        global vpPlaceStack2= pose_trans (pStackOutBase2_p, p[0,0,-1*iStackOut2*fSampleDoneZ,0,0,0])
        $ 1379 "PlaceStackOut"
        $ 1380 "If iStackOut1≤iStackOut2"
        if (iStackOut1 <= iStackOut2):
          $ 1381 "StackOut1"
          $ 1382 "vpTargetPos≔pose_trans(vpPlaceStack1, p[0,0,-5/1000,0,0,0])"
          global vpTargetPos= pose_trans (vpPlaceStack1, p[0,0,-5/1000,0,0,0])
          $ 1383 "MoveL"
          $ 1384 "pStackOut1Abv" "breakAfter"
          set_tcp(p[0.0,0.0,0.24273,0.0,0.0,-1.5708])
          movel(pStackOut1Abv_p, a=1.2, v=0.25, r=0.001)
          $ 1387 "MoveL"
          $ 1388 "vpTargetPos" "breakAfter"
          movel(vpTargetPos, a=2.5, v=0.75)
          $ 1389 "GripperOff()"
          GripperOff()
          $ 1390 "If bManualControl"
          if (bManualControl):
            $ 1391 "iStackOut1≔iStackOut1+1"
            global iStackOut1=iStackOut1+1
          end
          $ 1392 "vpTargetPos≔pose_trans(vpPlaceStack1, p[0,0,-25/1000,0,0,0])"
          global vpTargetPos= pose_trans (vpPlaceStack1, p[0,0,-25/1000,0,0,0])
          $ 1393 "MoveL"
          $ 1394 "vpTargetPos" "breakAfter"
          movel(vpTargetPos, a=1.2, v=0.25)
          $ 1395 "GripperOn()"
          GripperOn()
          $ 1396 "MoveL"
          $ 1397 "pStackOut1Abv" "breakAfter"
          movel(pStackOut1Abv_p, a=1.2, v=0.25)
        else:
          $ 1398 "Else" "noBreak"
          $ 1399 "StackOut2"
          $ 1400 "vpTargetPos≔pose_trans(vpPlaceStack2, p[0,0,-5/1000,0,0,0])"
          global vpTargetPos= pose_trans (vpPlaceStack2, p[0,0,-5/1000,0,0,0])
          $ 1401 "MoveJ"
          $ 1402 "pStackOut2Abv" "breakAfter"
          movej(get_inverse_kin(pStackOut2Abv_p, qnear=pStackOut2Abv_q), a=1.3962634015954636, v=1.0471975511965976)
          $ 1403 "MoveL"
          $ 1404 "vpTargetPos" "breakAfter"
          movel(vpTargetPos, a=1.2, v=0.25)
          $ 1405 "GripperOff()"
          GripperOff()
          $ 1406 "If bManualControl"
          if (bManualControl):
            $ 1407 "iStackOut2≔iStackOut2+1"
            global iStackOut2=iStackOut2+1
          end
          $ 1408 "vpTargetPos≔pose_trans(vpPlaceStack2, p[0,0,-25/1000,0,0,0])"
          global vpTargetPos= pose_trans (vpPlaceStack2, p[0,0,-25/1000,0,0,0])
          $ 1409 "MoveL"
          $ 1410 "vpTargetPos" "breakAfter"
          movel(vpTargetPos, a=1.2, v=0.25)
          $ 1411 "GripperOn()"
          GripperOn()
          $ 1412 "MoveL"
          $ 1413 "pStackOut2Abv" "breakAfter"
          movel(pStackOut2Abv_p, a=1.2, v=0.25)
          $ 1414 "pStackOutAbv" "breakAfter"
          movel(pStackOutAbv_p, a=1.2, v=0.25)
        end
        $ 1415 "Comment"
        # Comment
        $ 1416 "MoveJ"
        $ 1417 "pHomeTransit" "breakAfter"
        movej(get_inverse_kin(pHomeTransit_p, qnear=pHomeTransit_q), a=13.089969389957473, v=3.141592653589793, r=0.05)
        $ 1418 "pHome" "breakAfter"
        movej(get_inverse_kin(pHome_p, qnear=pHome_q), a=13.089969389957473, v=3.141592653589793)
        $ 1419 "iCycle≔iCycle-1"
        global iCycle=iCycle-1
      end
    else:
      $ 1648 "Default Case"
      $ 1649 "Comment"
      # Comment
    end
    $ 1650 "AssignFinishedState"
    $ 1651 "iStateOut≔iStateIn"
    global iStateOut=iStateIn
    $ 1652 "If iStateOut≠0"
    if (iStateOut != 0):
      $ 1653 "iLastState≔iStateOut"
      global iLastState=iStateOut
    end
    $ 1654 "If  not bManualControl"
    if (  not  bManualControl):
      $ 1655 "Wait iStateIn≠iStateOut"
      while (not(iStateIn != iStateOut)):
        sync()
      end
    end
    $ 1656 "sync()"
    sync()
  end
end
